// Implicitly generated code : DO NOT EDIT
FUNCTION CheckDivDInt : DINT
VAR_INPUT
	divisor:DINT;
END_VAR

// Implicitly generated code : Only an Implementation suggestion
{noflow}
IF divisor = 0 THEN
	GVL_Checks.diCheckDivDInt := GVL_Checks.diCheckDivDInt +1;
	CheckDivDInt:=1;
ELSE
	CheckDivDInt:=divisor;
END_IF;
{flow}

END_FUNCTION

(* stored: Version 1.1.0.1, ProductVersion 3.1.4024.12
   POU CheckDivDInt: Id {ce16ce50-baf2-44cb-87fe-6dc84883bc38}, SpecialFunc CheckDivInt32 *)
